Fanuc TP program (LS listing): RESET_MOVE_SELECTION.LS

/PROG  RESET_MOVE_SELECTION
/ATTR
OWNER		= MNEDITOR;
COMMENT		= "ClearSelectReg";
PROG_SIZE	= 202;
CREATE		= DATE 26-06-26  TIME 13:06:54;
MODIFIED	= DATE 26-07-09  TIME 10:39:00;
FILE_NAME	= ;
VERSION		= 0;
LINE_COUNT	= 4;
MEMORY_SIZE	= 558;
PROTECT		= READ_WRITE;
TCD:  STACK_SIZE	= 0,
      TASK_PRIORITY	= 50,
      TIME_SLICE	= 0,
      BUSY_LAMP_OFF	= 0,
      ABORT_REQUEST	= 0,
      PAUSE_REQUEST	= 0;
DEFAULT_GROUP	= *,*,*,*,*;
CONTROL_CODE	= 00000000 00000000;
LOCAL_REGISTERS	= 0,0,0;
/MN
   1:   ;
   2:  !Reset selected cell register ;
   3:  R[13:SELECTED_CELL]=0    ;
   4:   ;
/POS
/END
